// TIA Portal V20 export
// export: Created 2026-04-28T10:17:59.0556665Z, ExportSetting WithDefaults, DisplayName Totally Integrated Automation Portal, DisplayVersion V20, DisplayName TIA Portal Openness, DisplayVersion V20, DisplayName TIA Portal Version Control Interface, DisplayVersion V20, DisplayName SINAMICS Startdrive Advanced, DisplayVersion V20, DisplayName SINAMICS Startdrive G130, G150, S120, S150, SINAMICS MV, G220, S200, S210, DisplayVersion V20, DisplayName SINAMICS Startdrive G110M, G120, G120C, G120D, G120P, G115D, DisplayVersion V20, DisplayName STEP 7 Professional, DisplayVersion V20, DisplayName STEP 7 Safety, DisplayVersion V20, DisplayName WinCC Basic/Comfort/Advanced, DisplayVersion V20, DisplayName WinCC Unified, DisplayVersion V20
TYPE "Daten_SPT_30"
// stored: IsFailsafeCompliant false
   STRUCT
      xRiddle : Bool := false;   // Selection Riddle
      xCoBelt : Bool := false;   // Selection Conveyor belt
      xViCo1 : Bool := false;   // Selection Vibrating trough
      xReGrHu : Bool := false;   // Selection Resedual granulate humidity
      RangeReGrHu : DInt := 0;   // Residual granulate humidity range
      txt_rReGrHuMa : DInt := 0;   // Residual granulate humidity max.
      txt_max_rReGrHuMa : DInt := 0;   // Residual granulate humidity max.
      xReGrHuReg : Bool := false;   // Selection Residual humidity control
      txt_rReGrHuSoll : DInt := 0;   // Residual granulate humidity Set Value
      iTakt_ReGrHu : DInt := 0;   // Interval for recording the measured values
      iAnzWerte_ReGrH : DInt := 0;   // Number of measured values
      xGranulate : Bool := false;   // Selection Granulate
      xGrTe : Bool := false;   // Selection Granulate Temperature
      txt_rGrTeMa : DInt := 0;   // Granule temperature limit
      txt_max_rGrTeMa : DInt := 0;   // Granule temperature Input limit
      iTakt_GrTe : DInt := 0;   // Interval for recording the measured values
      iAnzWerte_GrTe : DInt := 0;   // Number of measured values
      xBarrel : Bool := false;   // Selection Barrel
      xScale : Bool := false;   // Selection Scale
      xFilling_1 : Bool := false;   // Selection Filling installaton 1
      txt_rEmpBin_1 : DInt := 0;   // Bin 1 empty
      txt_rFullBin_1 : DInt := 0;   // Bin 1 Full
      RangeScale_1 : DInt := 0;   // Range Scale 1
      txt_rWarn_1 : DInt := 0;   // Bin 1 Fill warning in %
      iTakt_1_Filling : DInt := 0;   // Interval for recording the measured values
      iAnzWerte_1_Fil : DInt := 0;   // Number of measured values
      xFilling_2 : Bool := false;   // Selection Filling installaton 2
      txt_rEmpBin_2 : DInt := 0;   // Bin 2 empty
      txt_rFullBin_2 : DInt := 0;   // Bin 2 Full
      RangeScale_2 : DInt := 0;   // Range Scale 2
      txt_rWarn_2 : DInt := 0;   // Bin 2 Fill warning in %
      iTakt_2_Filling : DInt := 0;   // Interval for recording the measured values
      iAnzWerte_2_Fil : DInt := 0;   // Number of measured values
      xTwPeVaTop : Bool := false;   // Selection Double pendulum flap 1
      t_iTwPeVaTopOp : Time := T#0MS;   // Double pendulum flap 1 open
      xTwPeVaBot : Bool := false;   // Selection Double pendulum flap 2
      t_iTwPeVaBotOp : Time := T#0MS;   // Double pendulum flap 2 open
      xGranulatSwitch : Bool := false;   // Selection Granulate switch
      xCoolWaterFlCo : Bool := false;   // Selection Cooling water flow monitor
      iTakt_CoWaFlCo : DInt := 0;   // Interval for recording the measured values
      iAnzW_CoWaFlCo : DInt := 0;   // Number of measured values
      RangeCoWaFlCo : DInt := 0;   // Range Cooling water flow monitor
      txt_CoWaFlCo : DInt := 0;   // Min. flow rate
      iTakt_CoWaTemp : DInt := 0;   // Interval for recording the measured values
      iAnzW_CoWaTemp : DInt := 0;   // Number of measured values
      RangeCoWaTemp : DInt := 0;   // Range cooling water temperature
      xFilling_OhneWaage : Bool := false;   // Filling installation 1 Without scale 1= Without scale with digital sensors
      xCoBelt_2 : Bool := false;   // Selection Conveyor belt 2.
      xFilling_5_LevelMes : Bool := false;   // Filling installation with 5 containers and analog level measurement 0=without, 1=with
      iTakt_LevelMes : DInt := 0;   // Interval for recording the measured values
      iAnzW_LevelMes : DInt := 0;   // Number of measured values
      RangeLevelMes : DInt := 0;   // Range level measurement
      xGrTeCtrl_Intervall : Bool := false;   // Selection Granulate Temperature monitoring at defined intervals
      txt_rGrTeCtrl_Up : DInt := 0;   // Selection Granulate Temperature monitoring at defined intervals Up
      txt_rGrTeCtrl_Down : DInt := 0;   // Selection Granulate Temperature monitoring at defined intervals Below
      xCtrlCoBelt_Option : Bool := false;   // Selection Conveyor belt monitoring rotation 0=without, 1=with
      xRidOverflow_Option : Bool;   // Selection Riddle overflow warning
      t_iPolyCoOn_ON : Time;   // Polyconveyor ON
      t_iPolyCoOn_OFF : Time;   // Polyconveyor OFF
      xPolyCoOn_Option : Bool;   // Selection Polyconveyor
      x_BinLevelMax_Option : Bool;   // Selection Buffer tank fill level max
      xPolyCoOn_2_Option : Bool;   // Selection Polyconveyor 2
      xUeberCOverflow_Option : Bool;   // Selection oversize container full
      t_iPumpeAus_TOF : Time;   // Delay switching off the polyf.
   END_STRUCT;
END_TYPE
